// TIA Portal V20 export
VAR_GLOBAL   // PLC tag table "Motors"
   STO_MST1 AT %Q357.0 : Bool;
   STO_MST38 AT %Q366.0 : Bool;
   STO_MST35 AT %Q264.0 : Bool;
   STO_MST34 AT %Q273.0 : Bool;
   STO_MST33a AT %Q282.0 : Bool;
   STO_MST33b AT %Q291.0 : Bool;
   STO_MST32 AT %Q327.0 : Bool;
   STO_MST31 AT %Q318.0 : Bool;
   STO_MST30a AT %Q336.0 : Bool;
   STO_MST36a AT %Q375.0 : Bool;
   STO_MST36b AT %Q384.0 : Bool;
   STO_MST37 AT %Q418.0 : Bool;
   STO_MST18 AT %Q437.0 : Bool;
   STO_MST19a AT %Q467.0 : Bool;
   STO_MST4a AT %Q486.0 : Bool;
   STO_MST4b AT %Q557.0 : Bool;
   STO_MST5 AT %Q576.0 : Bool;
   STO_MST6a AT %Q634.0 : Bool;
   STO_MST6b AT %Q667.0 : Bool;
   STO_MST7 AT %Q686.0 : Bool;
   STO_MST8 AT %Q705.0 : Bool;
   STO_MST9a AT %Q724.0 : Bool;
   STO_MST9b AT %Q743.0 : Bool;
   STO_MST10 AT %Q762.0 : Bool;
   STO_MST11 AT %Q781.0 : Bool;
   STO_MST12a AT %Q801.0 : Bool;
   STO_MST12b AT %Q820.0 : Bool;
   STO_MST13 AT %Q839.0 : Bool;
   STO_MST14 AT %Q858.0 : Bool;
   STO_MST17 AT %Q877.0 : Bool;
   STO_Mst19b AT %Q934.0 : Bool;
   STO_Mst20 AT %Q953.0 : Bool;
   STO_Mst21 AT %Q991.0 : Bool;
   STO_Mst22a AT %Q972.0 : Bool;
   STO_Mst22b AT %Q1010.0 : Bool;
   STO_Mst23a AT %Q1067.0 : Bool;
   STO_Mst23b AT %Q1029.0 : Bool;
   STO_Mst24a AT %Q1048.0 : Bool;
   STO_Mst24b AT %Q1086.0 : Bool;
   STO_MST1a AT %Q1131.0 : Bool;
   STO_Mst25a AT %Q1311.0 : Bool;
   STO_Mst25b AT %Q1330.0 : Bool;
   STO_Mst26 AT %Q1349.0 : Bool;
   STO_Mst27a AT %Q1368.0 : Bool;
   STO_Mst27b AT %Q1387.0 : Bool;
   STO_MST28 AT %Q1275.0 : Bool;
END_VAR
